// TIA Portal V17 export
// export: Created 2025-08-05T09:36:01.3929085Z, ExportSetting WithDefaults, DisplayName Totally Integrated Automation Portal, DisplayVersion V17, DisplayName TIA Portal Openness, DisplayVersion V17, DisplayName TIA Portal Version Control Interface, DisplayVersion V17, DisplayName SINAMICS Startdrive Advanced, DisplayVersion V17, DisplayName SINAMICS Startdrive G130, G150, S120, S150, SINAMICS MV, S210, DisplayVersion V17, DisplayName SINAMICS Startdrive G110M, G120, G120C, G120D, G120P, G115D, DisplayVersion V17, DisplayName STEP 7 Professional, DisplayVersion V17, DisplayName STEP 7 Safety, DisplayVersion V17, DisplayName WinCC Advanced, DisplayVersion V17
TYPE "typeKeyenceDetailedQuality"
// 01.00
// stored: IsFailsafeCompliant false
   STRUCT
      overall { ExternalAccessible := 'False'; ExternalVisible := 'False'; ExternalWritable := 'False'} : Char;   // Gesamtgüte / Overall quality
      overall_comma { ExternalAccessible := 'False'; ExternalVisible := 'False'; ExternalWritable := 'False'} : Char := ',';   // Komma / Comma
      dec { ExternalAccessible := 'False'; ExternalVisible := 'False'; ExternalWritable := 'False'} : Char;   // Deokdierung erfolgreich / fehlgeschlagen / Decoding successful / failed
      dec_comma { ExternalAccessible := 'False'; ExternalVisible := 'False'; ExternalWritable := 'False'} : Char := ',';   // Komma / Comma
      cc { ExternalAccessible := 'False'; ExternalVisible := 'False'; ExternalWritable := 'False'} : Char;   // Zellenkontrast / Cell contrast
      cc_comma { ExternalAccessible := 'False'; ExternalVisible := 'False'; ExternalWritable := 'False'} : Char := ',';   // Komma / Comma
      ccValue1 { ExternalAccessible := 'False'; ExternalVisible := 'False'; ExternalWritable := 'False'} : Char;   // Zellenkontrast (Wert) / Cell contrast (value)
      ccValue2 { ExternalAccessible := 'False'; ExternalVisible := 'False'; ExternalWritable := 'False'} : Char;   // Zellenkontrast (Wert) / Cell contrast (value)
      ccValue3 { ExternalAccessible := 'False'; ExternalVisible := 'False'; ExternalWritable := 'False'} : Char;   // Zellenkontrast (Wert) / Cell contrast (value)
      ccValue4 { ExternalAccessible := 'False'; ExternalVisible := 'False'; ExternalWritable := 'False'} : Char;   // Zellenkontrast (Wert) / Cell contrast (value)
      ccValue5 { ExternalAccessible := 'False'; ExternalVisible := 'False'; ExternalWritable := 'False'} : Char;   // Zellenkontrast (Wert) / Cell contrast (value)
      ccValue6 { ExternalAccessible := 'False'; ExternalVisible := 'False'; ExternalWritable := 'False'} : Char;   // Zellenkontrast (Wert) / Cell contrast (value)
      ccValue_comma { ExternalAccessible := 'False'; ExternalVisible := 'False'; ExternalWritable := 'False'} : Char := ',';   // Komma / Comma
      cm { ExternalAccessible := 'False'; ExternalVisible := 'False'; ExternalWritable := 'False'} : Char;   // Zellenmodulation / Cell modulation
      cm_comma { ExternalAccessible := 'False'; ExternalVisible := 'False'; ExternalWritable := 'False'} : Char := ',';   // Komma / Comma
      rm { ExternalAccessible := 'False'; ExternalVisible := 'False'; ExternalWritable := 'False'} : Char;   // Refelxtionsrand / Reflective edge
      rm_comma { ExternalAccessible := 'False'; ExternalVisible := 'False'; ExternalWritable := 'False'} : Char := ',';   // Komma / Comma
      fpd { ExternalAccessible := 'False'; ExternalVisible := 'False'; ExternalWritable := 'False'} : Char;   // Schäaden am festen Muster / Damage to the fixed sample
      fpd_comma { ExternalAccessible := 'False'; ExternalVisible := 'False'; ExternalWritable := 'False'} : Char := ',';   // Komma / Comma
      an { ExternalAccessible := 'False'; ExternalVisible := 'False'; ExternalWritable := 'False'} : Char;   // Axiale Verzerrung / Axial distortion
      an_comma { ExternalAccessible := 'False'; ExternalVisible := 'False'; ExternalWritable := 'False'} : Char := ',';   // Komma / Comma
      anValue1 { ExternalAccessible := 'False'; ExternalVisible := 'False'; ExternalWritable := 'False'} : Char;   // Axiale Verzerrung (Wert) / Axial distortion (value)
      anValue2 { ExternalAccessible := 'False'; ExternalVisible := 'False'; ExternalWritable := 'False'} : Char;   // Axiale Verzerrung (Wert) / Axial distortion (value)
      anValue3 { ExternalAccessible := 'False'; ExternalVisible := 'False'; ExternalWritable := 'False'} : Char;   // Axiale Verzerrung (Wert) / Axial distortion (value)
      anValue4 { ExternalAccessible := 'False'; ExternalVisible := 'False'; ExternalWritable := 'False'} : Char;   // Axiale Verzerrung (Wert) / Axial distortion (value)
      anValue5 { ExternalAccessible := 'False'; ExternalVisible := 'False'; ExternalWritable := 'False'} : Char;   // Axiale Verzerrung (Wert) / Axial distortion (value)
      anValue6 { ExternalAccessible := 'False'; ExternalVisible := 'False'; ExternalWritable := 'False'} : Char;   // Axiale Verzerrung (Wert) / Axial distortion (value)
      anValue_comma { ExternalAccessible := 'False'; ExternalVisible := 'False'; ExternalWritable := 'False'} : Char := ',';   // Komma / Comma
      gn { ExternalAccessible := 'False'; ExternalVisible := 'False'; ExternalWritable := 'False'} : Char;   // Rasterverzerrung / Grid distortion
      gn_comma { ExternalAccessible := 'False'; ExternalVisible := 'False'; ExternalWritable := 'False'} : Char := ',';   // Komma / Comma
      gnValue1 { ExternalAccessible := 'False'; ExternalVisible := 'False'; ExternalWritable := 'False'} : Char;   // Rasterverzerrung (Wert) / Grid distortion (value)
      gnValue2 { ExternalAccessible := 'False'; ExternalVisible := 'False'; ExternalWritable := 'False'} : Char;   // Rasterverzerrung (Wert) / Grid distortion (value)
      gnValue3 { ExternalAccessible := 'False'; ExternalVisible := 'False'; ExternalWritable := 'False'} : Char;   // Rasterverzerrung (Wert) / Grid distortion (value)
      gnValue4 { ExternalAccessible := 'False'; ExternalVisible := 'False'; ExternalWritable := 'False'} : Char;   // Rasterverzerrung (Wert) / Grid distortion (value)
      gnValue5 { ExternalAccessible := 'False'; ExternalVisible := 'False'; ExternalWritable := 'False'} : Char;   // Rasterverzerrung (Wert) / Grid distortion (value)
      gnValue6 { ExternalAccessible := 'False'; ExternalVisible := 'False'; ExternalWritable := 'False'} : Char;   // Rasterverzerrung (Wert) / Grid distortion (value)
      gnValue_comma { ExternalAccessible := 'False'; ExternalVisible := 'False'; ExternalWritable := 'False'} : Char := ',';   // Komma / Comma
      uec { ExternalAccessible := 'False'; ExternalVisible := 'False'; ExternalWritable := 'False'} : Char;   // Nicht verwendete Fehlerkorrektur / Unused error correction
      uec_comma { ExternalAccessible := 'False'; ExternalVisible := 'False'; ExternalWritable := 'False'} : Char := ',';   // Komma / Comma
      uecValue1 { ExternalAccessible := 'False'; ExternalVisible := 'False'; ExternalWritable := 'False'} : Char;   // Nicht verwendete Fehlerkorrektur (Wert) / Unused error correction (value)
      uecValue2 { ExternalAccessible := 'False'; ExternalVisible := 'False'; ExternalWritable := 'False'} : Char;   // Nicht verwendete Fehlerkorrektur (Wert) / Unused error correction (value)
      uecValue3 { ExternalAccessible := 'False'; ExternalVisible := 'False'; ExternalWritable := 'False'} : Char;   // Nicht verwendete Fehlerkorrektur (Wert) / Unused error correction (value)
      uecValue4 { ExternalAccessible := 'False'; ExternalVisible := 'False'; ExternalWritable := 'False'} : Char;   // Nicht verwendete Fehlerkorrektur (Wert) / Unused error correction (value)
      uecValue5 { ExternalAccessible := 'False'; ExternalVisible := 'False'; ExternalWritable := 'False'} : Char;   // Nicht verwendete Fehlerkorrektur (Wert) / Unused error correction (value)
      uecValue6 { ExternalAccessible := 'False'; ExternalVisible := 'False'; ExternalWritable := 'False'} : Char;   // Nicht verwendete Fehlerkorrektur (Wert) / Unused error correction (value)
      uecValue_comma { ExternalAccessible := 'False'; ExternalVisible := 'False'; ExternalWritable := 'False'} : Char := ',';   // Komma / Comma
      fid { ExternalAccessible := 'False'; ExternalVisible := 'False'; ExternalWritable := 'False'} : Char;   // Schaden an Formatdaten / Damage to format data
      fid_comma { ExternalAccessible := 'False'; ExternalVisible := 'False'; ExternalWritable := 'False'} : Char := ',';   // Komma / Comma
      fidValue1 { ExternalAccessible := 'False'; ExternalVisible := 'False'; ExternalWritable := 'False'} : Char;   // Schaden an Formatdaten (Wert) / Damage to format data (value)
      fidValue2 { ExternalAccessible := 'False'; ExternalVisible := 'False'; ExternalWritable := 'False'} : Char;   // Schaden an Formatdaten (Wert) / Damage to format data (value)
      fidValue3 { ExternalAccessible := 'False'; ExternalVisible := 'False'; ExternalWritable := 'False'} : Char;   // Schaden an Formatdaten (Wert) / Damage to format data (value)
      fidValue4 { ExternalAccessible := 'False'; ExternalVisible := 'False'; ExternalWritable := 'False'} : Char;   // Schaden an Formatdaten (Wert) / Damage to format data (value)
      fidValue5 { ExternalAccessible := 'False'; ExternalVisible := 'False'; ExternalWritable := 'False'} : Char;   // Schaden an Formatdaten (Wert) / Damage to format data (value)
      fidValue6 { ExternalAccessible := 'False'; ExternalVisible := 'False'; ExternalWritable := 'False'} : Char;   // Schaden an Formatdaten (Wert) / Damage to format data (value)
      fidValue_comma { ExternalAccessible := 'False'; ExternalVisible := 'False'; ExternalWritable := 'False'} : Char := ',';   // Komma / Comma
      vid { ExternalAccessible := 'False'; ExternalVisible := 'False'; ExternalWritable := 'False'} : Char;   // Modelldatenschaden / Model data damage
      vid_comma { ExternalAccessible := 'False'; ExternalVisible := 'False'; ExternalWritable := 'False'} : Char := ',';   // Komma / Comma
      vidValue1 { ExternalAccessible := 'False'; ExternalVisible := 'False'; ExternalWritable := 'False'} : Char;   // Modelldatenschaden (Wert) / Model data damage (value)
      vidValue2 { ExternalAccessible := 'False'; ExternalVisible := 'False'; ExternalWritable := 'False'} : Char;   // Modelldatenschaden (Wert) / Model data damage (value)
      vidValue3 { ExternalAccessible := 'False'; ExternalVisible := 'False'; ExternalWritable := 'False'} : Char;   // Modelldatenschaden (Wert) / Model data damage (value)
      vidValue4 { ExternalAccessible := 'False'; ExternalVisible := 'False'; ExternalWritable := 'False'} : Char;   // Modelldatenschaden (Wert) / Model data damage (value)
      vidValue5 { ExternalAccessible := 'False'; ExternalVisible := 'False'; ExternalWritable := 'False'} : Char;   // Modelldatenschaden (Wert) / Model data damage (value)
      vidValue6 { ExternalAccessible := 'False'; ExternalVisible := 'False'; ExternalWritable := 'False'} : Char;   // Modelldatenschaden (Wert) / Model data damage (value)
      vidValue_comma { ExternalAccessible := 'False'; ExternalVisible := 'False'; ExternalWritable := 'False'} : Char := ',';   // Komma / Comma
      pgh { ExternalAccessible := 'False'; ExternalVisible := 'False'; ExternalWritable := 'False'} : Char;   // Druckskalierung horizontal / Print scaling horizontal
      pgh_comma { ExternalAccessible := 'False'; ExternalVisible := 'False'; ExternalWritable := 'False'} : Char := ',';   // Komma / Comma
      pghValue1 { ExternalAccessible := 'False'; ExternalVisible := 'False'; ExternalWritable := 'False'} : Char;   // Druckskalierung horizontal (Wert) / Print scaling horizontal (value)
      pghValue2 { ExternalAccessible := 'False'; ExternalVisible := 'False'; ExternalWritable := 'False'} : Char;   // Druckskalierung horizontal (Wert) / Print scaling horizontal (value)
      pghValue3 { ExternalAccessible := 'False'; ExternalVisible := 'False'; ExternalWritable := 'False'} : Char;   // Druckskalierung horizontal (Wert) / Print scaling horizontal (value)
      pghValue4 { ExternalAccessible := 'False'; ExternalVisible := 'False'; ExternalWritable := 'False'} : Char;   // Druckskalierung horizontal (Wert) / Print scaling horizontal (value)
      pghValue5 { ExternalAccessible := 'False'; ExternalVisible := 'False'; ExternalWritable := 'False'} : Char;   // Druckskalierung horizontal (Wert) / Print scaling horizontal (value)
      pghValue6 { ExternalAccessible := 'False'; ExternalVisible := 'False'; ExternalWritable := 'False'} : Char;   // Druckskalierung horizontal (Wert) / Print scaling horizontal (value)
      pghValue_comma { ExternalAccessible := 'False'; ExternalVisible := 'False'; ExternalWritable := 'False'} : Char := ',';   // Komma / Comma
      pgv { ExternalAccessible := 'False'; ExternalVisible := 'False'; ExternalWritable := 'False'} : Char;   // Druckskalierung vertikal / Print scaling vertical
      pgv_comma { ExternalAccessible := 'False'; ExternalVisible := 'False'; ExternalWritable := 'False'} : Char := ',';   // Komma / Comma
      pgvValue1 { ExternalAccessible := 'False'; ExternalVisible := 'False'; ExternalWritable := 'False'} : Char;   // Druckskalierung vertikal (Wert) / Print scaling vertical (value)
      pgvValue2 { ExternalAccessible := 'False'; ExternalVisible := 'False'; ExternalWritable := 'False'} : Char;   // Druckskalierung vertikal (Wert) / Print scaling vertical (value)
      pgvValue3 { ExternalAccessible := 'False'; ExternalVisible := 'False'; ExternalWritable := 'False'} : Char;   // Druckskalierung vertikal (Wert) / Print scaling vertical (value)
      pgvValue4 { ExternalAccessible := 'False'; ExternalVisible := 'False'; ExternalWritable := 'False'} : Char;   // Druckskalierung vertikal (Wert) / Print scaling vertical (value)
      pgvValue5 { ExternalAccessible := 'False'; ExternalVisible := 'False'; ExternalWritable := 'False'} : Char;   // Druckskalierung vertikal (Wert) / Print scaling vertical (value)
      pgvValue6 { ExternalAccessible := 'False'; ExternalVisible := 'False'; ExternalWritable := 'False'} : Char;   // Druckskalierung vertikal (Wert) / Print scaling vertical (value)
      pgvValue_comma { ExternalAccessible := 'False'; ExternalVisible := 'False'; ExternalWritable := 'False'} : Char := ',';   // Komma / Comma
   END_STRUCT;
END_TYPE
